TYPE EL1809_EX EXTENDS EL1809:
STRUCT
	WcState AT %I* : BOOL;
	InputToggle AT %I* : BOOL;
	State AT %I* : UINT;
END_STRUCT
END_TYPE

(* stored: Version 1.1.0.1, ProductVersion 3.1.4026.18
   DUT EL1809_EX: Id {a0369698-d9b3-40fb-98ce-8ad34b238c1d} *)
